{attribute addProperty BoxType "EJ5002-0000-0016"}
{attribute addProperty Id "SSI_Inputs_ChannelAT %I*ARRAY[0..2] OF SSI_Inputs_Channel_F7D238D196120WcStateAT %I*WcState_98A4DF7520.250InfoDataAT %I*InfoData_BC63D37F80100"}
{attribute addProperty CRC "3035886411"}
{attribute addProperty SizeInBites "178"}
{attribute addProperty SizeInBytes "22.25"}
TYPE EJ5002_82283068 :
STRUCT
	{attribute addProperty Name "SSI_Inputs_Channel"}
	SSI_Inputs_Channel : ARRAY[0..2] OF SSI_Inputs_Channel_F7D238D1;
	{attribute addProperty Name "WcState"}
	WcState : WcState_98A4DF75;
	{attribute addProperty Name "InfoData"}
	InfoData : InfoData_BC63D37F;
END_STRUCT
END_TYPE

(* stored: Version 1.2.0.0, ProductVersion 3.1.4024.9
   DUT EJ5002_82283068: Id {810546e4-dd84-43a9-9910-44b9f9a6a453} *)
